(******************************************************************************
Baustein: PRG_TestLibrary
Spezifikation: doc/Spezifikation.pdf, Kap. x.y.z
-------------------------------------------------------------------------------
erstellt:
von:
Geändert:
von:
-------------------------------------------------------------------------------
Beschreibung
Dieser Baustein etnhält alle Testsuites und führt diese aus.

-------------------------------------------------------------------------------
Input
	i_bStart : mit positiver Flanke werden die registrierten Testsuites ausgeführt

Output
	o_eState  		: EState_t;
	o_eResult 		: EResult_t;
	o_sStatistic	: SStatistic_t;
******************************************************************************)
{attribute 'global_init_slot' := '41000'}
PROGRAM PRG_TestCoverage
VAR_INPUT
	i_bStart : BOOL;
END_VAR
VAR_OUTPUT
	o_eState  		: EState_t;
	o_eResult 		: EResult_t;
	o_sStatistic	: SStatistic_t;
END_VAR
VAR


	pTestReport		: POINTER TO FB_TestReportBase;
	eRetCode 		: ERetCode_t;

	fbSystemTime 	: FB_LocalSystemTime;
	
	fbCoverage 		: FB_CoverageFile;

	u16PouIdx  		: UINT;
	u16LineIdx 		: UINT;
	u16ReportState  : UINT;
	sCodeCoverage	: SCodeCoverage_t;
	
END_VAR
VAR CONSTANT 
	u32MaxLineIdx   : UDINT := 2000; (* maximale Zeilenanzahl   *)
	u32MaxPouIdx    : UDINT := 500;  (* maximale Bausteinanzahl *)
END_VAR



	fbCoverage();
		
	CASE o_eState OF 
	
	EState_t.eStateIdle:	
		
		IF i_bStart = FALSE THEN 
		   logInfo('Testlib V1.1.1 Ready');
			o_eState := EState_t.eStateIdle; 
		END_IF
	
	EState_t.eStateExecute:
	
		IF createReport(EReporttype_t.eCoverageReport) = ERetCode_t.eRetDone THEN
			o_eState := EState_t.eStateReady;
		END_IF;
		
	EState_t.eStateReady:

		IF i_bStart  = FALSE THEN
			o_eState := EState_t.eStateIdle;
		END_IF		
		
	EState_t.eStateError,
	EState_t.eStateLicenseError:
	
		o_eState := EState_t.eStateError;

	END_CASE

{attribute 'hide'} 
METHOD PRIVATE createReport : ERetCode_t
VAR_INPUT
	i_eReporttype : EReportType_t;
END_VAR
VAR
	eRetcode : ERetCode_t;
	u32Temp : UDINT;
END_VAR

	createReport := ERetCode_t.eRetBusy;

	CASE u16ReportState OF

	0: 
		IF i_eReporttype = EReportType_t.eCoverageReport THEN
			u16ReportState := 10;
		END_IF;

// +++++++++++++++++++++++++++++++++++++++++++++++++++++++++++
//
// Export Codeabdeckung
// 
// +++++++++++++++++++++++++++++++++++++++++++++++++++++++++++
	10:
		eRetcode := fbCoverage.open('C:\TwinCAT\3.1\Boot\CurrentConfig\', 'Coverage.xml');

		IF eRetcode = ERetCode_t.eRetDone THEN

			u16ReportState := 11;

		ELSIF eRetcode = ERetCode_t.eRetFailed THEN

			logError('createReport Coverage.xml : Datei nicht geöffnet');
			u16ReportState := 12;

		END_IF;		

	11:

		fbCoverage.addString('<?xml version="1.0" ?>');
		fbCoverage.addCrlf();

		fbCoverage.addString('<Result>');
		fbCoverage.addCrlf();

		FOR u16PouIdx := 1 TO sCodeCoverage.u16MaxPouIndex DO

			fbCoverage.addString('<POU Id="');
			fbCoverage.addValue(u16PouIdx);
			fbCoverage.addString('">');
			fbCoverage.addCrlf();

			FOR u16LineIdx := 1 TO sCodeCoverage.u16MaxLineIndex DO

				IF sCodeCoverage.aPou[u16PouIdx][u16LineIdx] > 0 THEN

					fbCoverage.addString('<Line Nb="');
					fbCoverage.addValue(u16LineIdx);

					fbCoverage.addString('" Count="');
					fbCoverage.addValue(sCodeCoverage.aPou[u16PouIdx][u16LineIdx]);
					
					fbCoverage.addString('"/>');
					fbCoverage.addCrlf();

				END_IF;

			END_FOR;

			fbCoverage.addString('</POU>');
			fbCoverage.addCrlf();

		END_FOR;

		fbCoverage.addString('</Result>');
		fbCoverage.addCrlf();
		u16ReportState := 12;


	12:

		IF fbCoverage.o_bOpen  = TRUE AND 
		   fbCoverage.o_bEmpty = TRUE THEN
			fbCoverage.close();
		END_IF;

		IF fbCoverage.o_bOpen  = FALSE THEN
			createReport 	:= ERetCode_t.eRetDone;
		END_IF;

	ELSE
		createReport := ERetCode_t.eRetFailed;
	END_CASE;

	IF createReport = ERetCode_t.eRetDone THEN
		u16ReportState := 0;
	END_IF;
















(**)
END_METHOD

(******************************************************************************
Baustein: PRG_UnitTestLib.getTime
Spezifikation: doc/Spezifikation.pdf, Kap. x.y.z
-------------------------------------------------------------------------------
erstellt:
von:
Geändert:
von:
-------------------------------------------------------------------------------
Beschreibung
Diese Methode

-------------------------------------------------------------------------------
Input
-

Output
-
******************************************************************************)
{attribute 'hide'} 
METHOD getTime : TimeStruct
VAR_INPUT
END_VAR
VAR
END_VAR

	getTime := fbSystemTime.systemTime;
END_METHOD

{attribute 'hide'} 
METHOD PUBLIC LineCovered : BOOL
VAR_INPUT
	u16Pou  : UINT;
	u16Line : UINT;
END_VAR

  LineCovered := TRUE;
	
  IF (u16Pou  > 0 AND u16Pou  <= u32MaxPouIdx ) AND
		 (u16Line > 0 AND u16Line <= u32MaxLineIdx) THEN
  
	  IF u16Pou > sCodeCoverage.u16MaxPouIndex THEN
		  sCodeCoverage.u16MaxPouIndex := u16Pou;
	  END_IF;
	  IF u16Line > sCodeCoverage.u16MaxLineIndex THEN
		  sCodeCoverage.u16MaxLineIndex := u16Line;
	  END_IF;
	  
	  IF sCodeCoverage.aPou[u16Pou][u16Line] < 255 THEN
		  sCodeCoverage.aPou[u16Pou][u16Line] := sCodeCoverage.aPou[u16Pou][u16Line]+1;
	  END_IF;
  END_IF;
END_METHOD

(******************************************************************************
Baustein: PRG_UnitTestLib.logError
Spezifikation: doc/Spezifikation.pdf, Kap. x.y.z
-------------------------------------------------------------------------------
erstellt:
von:
Geändert:
von:
-------------------------------------------------------------------------------
Beschreibung
Diese Methode

-------------------------------------------------------------------------------
Input
i_strMessage

Output
-
******************************************************************************)
{attribute 'hide'} 
METHOD PROTECTED logError : BOOL
VAR_INPUT
	i_strMessage : StrMessage_t;
END_VAR

	ADSLOGSTR(msgCtrlMask 	:= ADSLOG_MSGTYPE_ERROR , 
			  msgFmtStr 	:= i_strMessage, 
			  strArg 		:= '');
END_METHOD

(******************************************************************************
Baustein: PRG_UnitTestLib.logInfo
Spezifikation: doc/Spezifikation.pdf, Kap. x.y.z
-------------------------------------------------------------------------------
erstellt:
von:
Geändert:
von:
-------------------------------------------------------------------------------
Beschreibung
Diese Methode

-------------------------------------------------------------------------------
Input
i_strMessage

Output
-
******************************************************************************)
{attribute 'hide'} 
METHOD PUBLIC logInfo : BOOL
VAR_INPUT
	i_strMessage : StrMessage_t;
END_VAR

	ADSLOGSTR(msgCtrlMask 	:= ADSLOG_MSGTYPE_HINT , 
			  msgFmtStr 	:= i_strMessage, 
			  strArg 		:= '');
END_METHOD

END_PROGRAM

(* stored: Version 1.1.0.1, ProductVersion 3.1.4024.9
   POU PRG_TestCoverage: Id {89411254-1a6b-4317-931a-d4bd0576cd2f}, SpecialFunc None
   Method createReport: Id {edd1de35-26e0-498e-8636-7e4054f50d82}
   Method getTime: Id {fe4cca3a-6c07-4982-9c1c-91c2c139ab04}
   Method LineCovered: Id {a6330277-f233-45b1-ab10-e30e40611447}
   Method logError: Id {b61ecc79-d71a-4298-a53e-ef31f447bae7}
   Method logInfo: Id {9d54e29d-5872-467f-a5be-c4c4f1bef70e} *)
